PROGRAM MAIN
VAR
	Test	: BOOL := FALSE;
	i		: INT;
END_VAR


i := i + 1;


IF Test THEN
	
	Tests();
	
ELSE
	
	Application();
	
END_IF

Utility();

END_PROGRAM

(* stored: Version 1.1.0.1
   POU MAIN: Id {85dee3db-2224-4778-955d-df7bd8df7b99}, SpecialFunc None *)
